{attribute addProperty BoxType "EL3204-0000-0017"}
{attribute addProperty Id "RTD_Inputs_ChannelAT %I*ARRAY[0..6] OF RTD_Inputs_Channel_B51B79FC32440.50WcStateAT %I*WcState_98A4DF7520.250InfoDataAT %I*InfoData_BC63D37F80100"}
{attribute addProperty CRC "1598045051"}
{attribute addProperty SizeInBites "406"}
{attribute addProperty SizeInBytes "50.75"}
TYPE EL3204_C7F08A94 :
STRUCT
	{attribute addProperty Name "RTD_Inputs_Channel"}
	RTD_Inputs_Channel : ARRAY[0..6] OF RTD_Inputs_Channel_B51B79FC;
	{attribute addProperty Name "WcState"}
	WcState : WcState_98A4DF75;
	{attribute addProperty Name "InfoData"}
	InfoData : InfoData_BC63D37F;
END_STRUCT
END_TYPE

(* stored: Version 1.2.0.0, ProductVersion 3.1.4024.9
   DUT EL3204_C7F08A94: Id {cf4ecfd8-b29a-4974-afdf-148656ab483d} *)
